TYPE sysTimersCounters :
STRUCT
	
	doorOpenTimer : TON;
	doorCloseTimer : TON;
	rpiPingTimer : TON;
	rpiWaitTimer : TON;


	testButtonTimer : TON;
	alarmButtonTImer : TON; 
	alarmButtonTimer_HMI : TON;
	testButtonTimer_HMI  : TON;

	
	
END_STRUCT

END_TYPE

(* stored: Version 1.1.0.1, ProductVersion 3.1.4026.12
   DUT sysTimersCounters: Id {54b2a0a0-2e71-4e07-b7fc-0eb31cc25951} *)
